FUNCTION_BLOCK FB_Ramp
VAR_INPUT
	start	: INT;
	target	: INT;
	accel	: UINT;
END_VAR
VAR_OUTPUT
	value	: INT;
END_VAR
VAR
END_VAR

value := start;

// step
// compare in DINT: a reversal (e.g. -30000 -> +30000) does not fit in 16 bit
IF TO_DINT(target) - TO_DINT(value) > 0 THEN	
	value := value + TO_INT(accel);
	IF value >= target THEN
		value := target;
	END_IF
ELSE
	value := value - TO_INT(accel);
	IF value <= target THEN
		value := target;
	END_IF
END_IF

END_FUNCTION_BLOCK

(* stored: Version 1.1.0.1, ProductVersion 3.1.4024.15
   POU FB_Ramp: Id {4c8732d7-c459-4056-a387-72e8aeca0bce}, SpecialFunc None *)
